DATA_BLOCK "local_control"
{ S7_Optimized_Access := 'FALSE' }
VERSION : 0.1
   STRUCT
      start_stop : Array[0..5] of Bool;
      pump_maintain : Array[0..5] of Bool;
      flow_set : Array[0..5] of Real;
      flow_read : Array[0..5] of Real;
      tank_level : Array[0..5] of Real;
      valve_action : Array[0..5] of Bool;
      low_level_alarm : Array[0..5] of Bool;
      low_level_alarm_set : Array[0..5] of Real;
      flow_meter_read : Array[0..50] of Bool;
      flow_meter_read_error : Array[0..5] of Word;
      dosing_flow : Array[0..20] of Real;
      dosing_accumulate : Array[0..20] of Real;
      valve_opening : Array[0..5] of Bool;
      valve_closing : Array[0..5] of Bool;
      high_level_alarm : Array[0..5] of Bool;
      high_level_alarm_set : Array[0..5] of Real;
      energy_meter : Array[0..10] of Real;
      tank_weigh : Array[0..5] of Real;
      low_flow_alarm_set : Array[0..10] of Real;
      low_flow_alarm : Array[0..10] of Bool;
   END_STRUCT;


BEGIN

END_DATA_BLOCK

